FUNCTION F_Concat3 : String
VAR_INPUT
	sString1 : STRING;
	sString2 : STRING;
	sString3 : STRING;
END_VAR
VAR
END_VAR

F_Concat3 := CONCAT(F_Concat3, sString1);
F_Concat3 := CONCAT(F_Concat3, sString2);
F_Concat3 := CONCAT(F_Concat3, sString3);

END_FUNCTION

(* stored: Version 1.1.0.1, ProductVersion 3.1.4022.18
   POU F_Concat3: Id {f7fdd798-9cbc-42fc-89c6-f6302fb459d0}, SpecialFunc None *)
